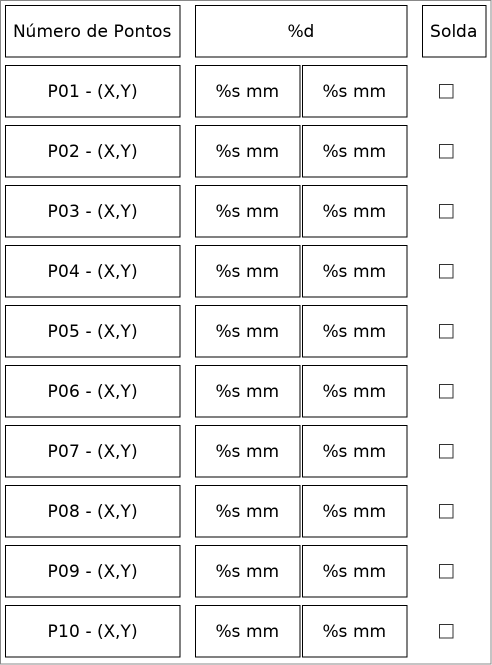
VISUALIZATION Lista_Receita_1  // 492x665
    Rectangle (5,5 175x52), "Número de Pontos"
    Rectangle (195,5 212x52), "%d", text variable: Recipe_N_Pontos_Solda, input disabled if: Not b_editar_receita and Not b_criar_receita
        OnMouseClick: write the text variable via Default
    Rectangle (5,65 175x52), "P01 - (X,Y)", invisible if: Recipe_N_Pontos_Solda<1
    Rectangle (195,65 105x52), "%s mm", text variable: Recipe_P_X01_Solda_Select, invisible if: Recipe_N_Pontos_Solda<1, input disabled if: Not b_editar_receita and Not b_criar_receita
        OnMouseClick: write the text variable via Default, min 0, max 300
    Rectangle (5,125 175x52), "P02 - (X,Y)", invisible if: Recipe_N_Pontos_Solda<2
    Rectangle (195,125 105x52), "%s mm", text variable: Recipe_P_X02_Solda_Select, invisible if: Recipe_N_Pontos_Solda<2, input disabled if: Not b_editar_receita and Not b_criar_receita
        OnMouseClick: write the text variable via Default
    Rectangle (5,185 175x52), "P03 - (X,Y)", invisible if: Recipe_N_Pontos_Solda<3
    Rectangle (195,185 105x52), "%s mm", text variable: Recipe_P_X03_Solda_Select, invisible if: Recipe_N_Pontos_Solda<3, input disabled if: Not b_editar_receita and Not b_criar_receita
        OnMouseClick: write the text variable via Default
    Rectangle (5,245 175x52), "P04 - (X,Y)", invisible if: Recipe_N_Pontos_Solda<4
    Rectangle (195,245 105x52), "%s mm", text variable: Recipe_P_X04_Solda_Select, invisible if: Recipe_N_Pontos_Solda<4, input disabled if: Not b_editar_receita and Not b_criar_receita
        OnMouseClick: write the text variable via Default
    Rectangle (5,305 175x52), "P05 - (X,Y)", invisible if: Recipe_N_Pontos_Solda<5
    Rectangle (195,305 105x52), "%s mm", text variable: Recipe_P_X05_Solda_Select, invisible if: Recipe_N_Pontos_Solda<5, input disabled if: Not b_editar_receita and Not b_criar_receita
        OnMouseClick: write the text variable via Default
    Rectangle (302,65 105x52), "%s mm", text variable: Recipe_P_Y01_Solda_Select, invisible if: Recipe_N_Pontos_Solda<1, input disabled if: Not b_editar_receita and Not b_criar_receita
        OnMouseClick: write the text variable via Default
    Rectangle (302,125 105x52), "%s mm", text variable: Recipe_P_Y02_Solda_Select, invisible if: Recipe_N_Pontos_Solda<2, input disabled if: Not b_editar_receita and Not b_criar_receita
        OnMouseClick: write the text variable via Default
    Rectangle (302,185 105x52), "%s mm", text variable: Recipe_P_Y03_Solda_Select, invisible if: Recipe_N_Pontos_Solda<3, input disabled if: Not b_editar_receita and Not b_criar_receita
        OnMouseClick: write the text variable via Default
    Rectangle (302,245 105x52), "%s mm", text variable: Recipe_P_Y04_Solda_Select, invisible if: Recipe_N_Pontos_Solda<4, input disabled if: Not b_editar_receita and Not b_criar_receita
        OnMouseClick: write the text variable via Default
    Rectangle (302,305 105x52), "%s mm", text variable: Recipe_P_Y05_Solda_Select, invisible if: Recipe_N_Pontos_Solda<5, input disabled if: Not b_editar_receita and Not b_criar_receita
        OnMouseClick: write the text variable via Default
    Rectangle (422,5 64x52), "Solda"
    Checkbox (437,71 40x40), variable: Recipe_P01_Solda_Select, invisible if: Recipe_N_Pontos_Solda<1, input disabled if: Not b_editar_receita and Not b_criar_receita
    Checkbox (437,131 40x40), variable: Recipe_P02_Solda_Select, invisible if: Recipe_N_Pontos_Solda<2, input disabled if: Not b_editar_receita and Not b_criar_receita
    Checkbox (437,191 40x40), variable: Recipe_P03_Solda_Select, invisible if: Recipe_N_Pontos_Solda<3, input disabled if: Not b_editar_receita and Not b_criar_receita
    Checkbox (437,251 40x40), variable: Recipe_P04_Solda_Select, invisible if: Recipe_N_Pontos_Solda<4, input disabled if: Not b_editar_receita and Not b_criar_receita
    Checkbox (437,311 40x40), variable: Recipe_P05_Solda_Select, invisible if: Recipe_N_Pontos_Solda<5, input disabled if: Not b_editar_receita and Not b_criar_receita
    Rectangle (5,365 175x52), "P06 - (X,Y)", invisible if: Recipe_N_Pontos_Solda<6
    Rectangle (195,365 105x52), "%s mm", text variable: Recipe_P_X06_Solda_Select, invisible if: Recipe_N_Pontos_Solda<6, input disabled if: Not b_editar_receita and Not b_criar_receita
        OnMouseClick: write the text variable via Default
    Rectangle (5,425 175x52), "P07 - (X,Y)", invisible if: Recipe_N_Pontos_Solda<7
    Rectangle (195,425 105x52), "%s mm", text variable: Recipe_P_X07_Solda_Select, invisible if: Recipe_N_Pontos_Solda<7, input disabled if: Not b_editar_receita and Not b_criar_receita
        OnMouseClick: write the text variable via Default
    Rectangle (5,485 175x52), "P08 - (X,Y)", invisible if: Recipe_N_Pontos_Solda<8
    Rectangle (195,485 105x52), "%s mm", text variable: Recipe_P_X08_Solda_Select, invisible if: Recipe_N_Pontos_Solda<8, input disabled if: Not b_editar_receita and Not b_criar_receita
        OnMouseClick: write the text variable via Default
    Rectangle (5,545 175x52), "P09 - (X,Y)", invisible if: Recipe_N_Pontos_Solda<9
    Rectangle (195,545 105x52), "%s mm", text variable: Recipe_P_X09_Solda_Select, invisible if: Recipe_N_Pontos_Solda<9, input disabled if: Not b_editar_receita and Not b_criar_receita
        OnMouseClick: write the text variable via Default
    Rectangle (5,605 175x52), "P10 - (X,Y)", invisible if: Recipe_N_Pontos_Solda<10
    Rectangle (195,605 105x52), "%s mm", text variable: Recipe_P_X10_Solda_Select, invisible if: Recipe_N_Pontos_Solda<10, input disabled if: Not b_editar_receita and Not b_criar_receita
        OnMouseClick: write the text variable via Default
    Rectangle (302,365 105x52), "%s mm", text variable: Recipe_P_Y06_Solda_Select, invisible if: Recipe_N_Pontos_Solda<6, input disabled if: Not b_editar_receita and Not b_criar_receita
        OnMouseClick: write the text variable via Default
    Rectangle (302,425 105x52), "%s mm", text variable: Recipe_P_Y07_Solda_Select, invisible if: Recipe_N_Pontos_Solda<7, input disabled if: Not b_editar_receita and Not b_criar_receita
        OnMouseClick: write the text variable via Default
    Rectangle (302,485 105x52), "%s mm", text variable: Recipe_P_Y08_Solda_Select, invisible if: Recipe_N_Pontos_Solda<8, input disabled if: Not b_editar_receita and Not b_criar_receita
        OnMouseClick: write the text variable via Default
    Rectangle (302,545 105x52), "%s mm", text variable: Recipe_P_Y09_Solda_Select, invisible if: Recipe_N_Pontos_Solda<9, input disabled if: Not b_editar_receita and Not b_criar_receita
        OnMouseClick: write the text variable via Default
    Rectangle (302,605 105x52), "%s mm", text variable: Recipe_P_Y10_Solda_Select, invisible if: Recipe_N_Pontos_Solda<10, input disabled if: Not b_editar_receita and Not b_criar_receita
        OnMouseClick: write the text variable via Default
    Checkbox (437,371 40x40), variable: Recipe_P06_Solda_Select, invisible if: Recipe_N_Pontos_Solda<6, input disabled if: Not b_editar_receita and Not b_criar_receita
    Checkbox (437,431 40x40), variable: Recipe_P07_Solda_Select, invisible if: Recipe_N_Pontos_Solda<7, input disabled if: Not b_editar_receita and Not b_criar_receita
    Checkbox (437,491 40x40), variable: Recipe_P08_Solda_Select, invisible if: Recipe_N_Pontos_Solda<8, input disabled if: Not b_editar_receita and Not b_criar_receita
    Checkbox (437,551 40x40), variable: Recipe_P09_Solda_Select, invisible if: Recipe_N_Pontos_Solda<9, input disabled if: Not b_editar_receita and Not b_criar_receita
    Checkbox (437,611 40x40), variable: Recipe_P10_Solda_Select, invisible if: Recipe_N_Pontos_Solda<10, input disabled if: Not b_editar_receita and Not b_criar_receita
END_VISUALIZATION

(* stored: Version 1.1.0.1, ProductVersion 3.1.4024.11
   Visu Lista_Receita_1: Id {ea5e6b0f-4800-48ff-a3b8-478b31d469c6} *)
